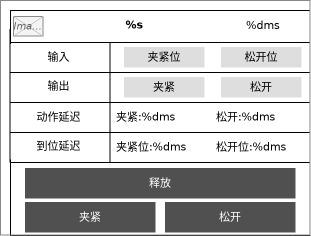
VISUALIZATION Cylinder5  // 311x236
VAR_INPUT
	System:							REFERENCE TO ST_System;
	Cylinder:						REFERENCE TO ST_Cylinder;
	CylinderData:					REFERENCE TO ST_CylinderData;
END_VAR
    RoundedRectangle (10,121 300x115)
    RoundedRectangle (10,10 300x115)
    Rectangle (10,44 300x115)
    Line (10,42) (310,42)
    Rectangle (45,13 179x24), "%s", text variable: Cylinder.arrInfo[System.stMode.eLanguage].sName, input disabled if: Cylinder.stLock.bShield
    Rectangle (228,13 70x25), "%dms", text variable: CylinderData.iAlarmTime, input disabled if: Cylinder.stLock.bShield
        OnMouseClick: write the text variable via VisuDialogs.Numpad
    Line (10,72) (310,72)
    Line (10,102) (310,102)
    Label (11,42 95x30), "输入"
    Label (11,71 95x30), "输出"
    Line (110,162) (110,42)
    RoundedRectangle (124,47 80x20), "夹紧位", colour toggle: Cylinder.stInput.bWork, input disabled if: Cylinder.stLock.bShield
    RoundedRectangle (221,47 80x20), "松开位", colour toggle: Cylinder.stInput.bHome, input disabled if: Cylinder.stLock.bShield
    RoundedRectangle (124,77 80x20), "夹紧", colour toggle: Cylinder.stOutput.bWork, input disabled if: Cylinder.stLock.bShield
    RoundedRectangle (221,77 80x20), "松开", colour toggle: Cylinder.stOutput.bHome, input disabled if: Cylinder.stLock.bShield
    RoundedRectangle (25,168 270x30), "释放", colour toggle: Cylinder.stLock.bOff OR Cylinder.stLock.bAll, input disabled if: Cylinder.stLock.bShield
        tap Cylinder.stControl.stOffRequest.bManual
    RoundedRectangle (25,202 130x30), "夹紧", colour toggle: Cylinder.stLock.bWork OR Cylinder.stLock.bAll, input disabled if: Cylinder.stLock.bShield
        tap Cylinder.stControl.stWorkRequest.bManual
    RoundedRectangle (165,202 130x30), "松开", colour toggle: Cylinder.stLock.bHome OR Cylinder.stLock.bAll, input disabled if: Cylinder.stLock.bShield
        tap Cylinder.stControl.stHomeRequest.bManual
    Line (310,164) (310,33)
    Line (10,162) (10,29)
    Image (13,16 30x20), image: ImagePool.Cylinder1
    Line (10,132) (310,132)
    Line (10,162) (310,162)
    Label (11,102 95x30), "动作延迟"
    Label (11,131 95x30), "到位延迟"
    RoundedRectangle (113,104 95x26), "夹紧:%dms", text variable: CylinderData.iWorkRequestTime, input disabled if: Cylinder.stLock.bShield
        OnMouseClick: write the text variable via Default
    RoundedRectangle (213,104 95x26), "松开:%dms", text variable: CylinderData.iHomeRequestTime, input disabled if: Cylinder.stLock.bShield
        OnMouseClick: write the text variable via Default
    RoundedRectangle (113,134 95x26), "夹紧位:%dms", text variable: CylinderData.iWorkDone, input disabled if: Cylinder.stLock.bShield
        OnMouseClick: write the text variable via Default
    RoundedRectangle (213,134 95x26), "松开位:%dms", text variable: CylinderData.iHomeDone, input disabled if: Cylinder.stLock.bShield
        OnMouseClick: write the text variable via Default
END_VISUALIZATION

(* stored: Version 1.1.0.1, ProductVersion 3.1.4024.4
   Visu Cylinder5: Id {3fae3928-1f70-464d-ab95-1b506872ebe9} *)
